FUNCTION_BLOCK CamInController
VAR_INPUT
	bExecute: BOOL;
	fSpeed : LREAL := 360;
END_VAR
VAR
	mcReset			: MC_Reset;
	mcPower			: MC_Power;
	mcStop			: MC_Stop;
	mcCamIn         : MC_CamIn;
	
	iState: UINT;;
END_VAR
VAR_IN_OUT
	Axis : AXIS_REF;
	Master : AXIS_REF;
END_VAR
VAR_OUTPUT
	bDone : BOOL;
END_VAR

mcReset(Axis:=Axis);
mcReset.Execute := FALSE;

mcPower(Axis:=Axis, Enable:=TRUE, Enable_Positive:=TRUE, Enable_Negative:=TRUE);

mcCamIn(Slave:=Axis, Master:= Master);
mcCamIn.Execute:=FALSE;

CASE iState OF
	0:	
		IF bExecute THEN
			iState:= 10;
		END_IF
		
	10: 
		// Reset the axis
		mcReset.Execute:=TRUE;
		iState := 20;
		bDone:= FALSE;
	
	20: 
		// Wait for reset to complete
		IF McReset.Done THEN
			iState := 30;
		ELSIF McReset.Error THEN
			iState := 999;
		END_IF
	
	30:
		// Set the power!
		IF McPower.Status THEN
			iState := 40;
		END_IF
		
	40:
		// Cam in
		mcCamIn.Execute:= TRUE;
		mcCamIn.SlaveScaling:= 1; 
		mcCamIn.CamTableID:= 1;
		
		iState:= 50;
	
	50: 
		// Done.
		IF mcCamIn.InSync THEN
			bDone := TRUE;
			iState := 0;
		END_IF
		
END_CASE

END_FUNCTION_BLOCK

(* stored: Version 1.1.0.1, ProductVersion 3.1.4022.10
   POU CamInController: Id {e44a4b46-4d0f-4a0e-8ad4-1de8ebcef60a}, SpecialFunc None *)
